(* Logix 5000 project; controller STAT 1756-L72 rev 20.12; software revision 20.04; part 18 of 34 *)
(* tags used below, declared in another part *)
   B14 : DINT[30];
   B16 : DINT[30];
   B17 : DINT[30];
   B3 : DINT[256];
   B9 : DINT[40];
   F8 : REAL[256];
   I1_005_Bit15 : ALIAS FOR I1[5].15;
   I6_001_Bit07 : ALIAS FOR I6[1].7;   // pulse debietmeter zandfilter osmose
   I7_000_Bit08 : ALIAS FOR I7[0].8;   // midden alarm ketel tampon
   N12 : DINT[230];
   N13 : DINT[230];
   N26 : DINT[256];
   O12_001_Bit14 : ALIAS FOR O12[1].14;   // STFA1_EV1 STFA1_EV1
   O12_001_Bit15 : ALIAS FOR O12[1].15;   // STFA1_EV2 STFA1_EV2
   O13_000_Bit00 : ALIAS FOR O13[0].0;   // STFA1_EV3 STFA1_EV3
   O13_000_Bit01 : ALIAS FOR O13[0].1;   // STFA1_EV4 STFA1_EV4
   O13_000_Bit02 : ALIAS FOR O13[0].2;   // STFA1_EV5 STFA1_EV5
   O13_000_Bit03 : ALIAS FOR O13[0].3;   // STFA1_EV6 STFA1_EV6
   O15_001_Bit13 : ALIAS FOR O15[1].13;   // TFB2_1_EV1 TFB2_1_EV1
   O15_001_Bit14 : ALIAS FOR O15[1].14;   // TFB2_1_EV2 TFB2_1_EV2
   O15_001_Bit15 : ALIAS FOR O15[1].15;   // TFB2_1_EV3 TFB2_1_EV3
   STEP_DUALM_3_4_5_6 : BOOL;
   STEP_NASPOEL_1_ET_2 : BOOL;
   T27 : TIMER[100];
   T4 : TIMER[200];
(* ibt, continued *)

ROUTINE _20_SEQ_VERZ1   (* ladder *)
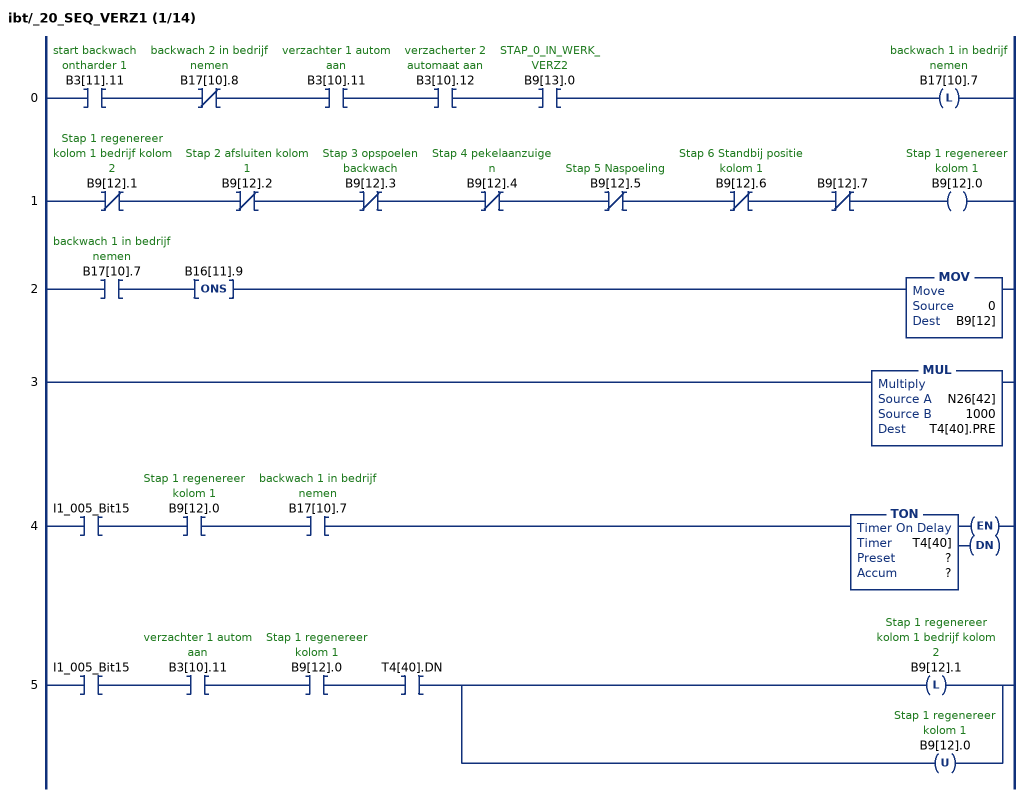
   0: XIC(B3[11].11)XIO(B17[10].8)XIC(B3[10].11)XIC(B3[10].12)XIC(B9[13].0)OTL(B17[10].7);
   1: XIO(B9[12].1)XIO(B9[12].2)XIO(B9[12].3)XIO(B9[12].4)XIO(B9[12].5)XIO(B9[12].6)XIO(B9[12].7)OTE(B9[12].0);
   2: XIC(B17[10].7)ONS(B16[11].9)MOV(0,B9[12]);
   3: MUL(N26[42],1000,T4[40].PRE);
   4: XIC(I1_005_Bit15)XIC(B9[12].0)XIC(B17[10].7)TON(T4[40],?,?);
   5: XIC(I1_005_Bit15)XIC(B3[10].11)XIC(B9[12].0)XIC(T4[40].DN)[OTL(B9[12].1) ,OTU(B9[12].0) ];
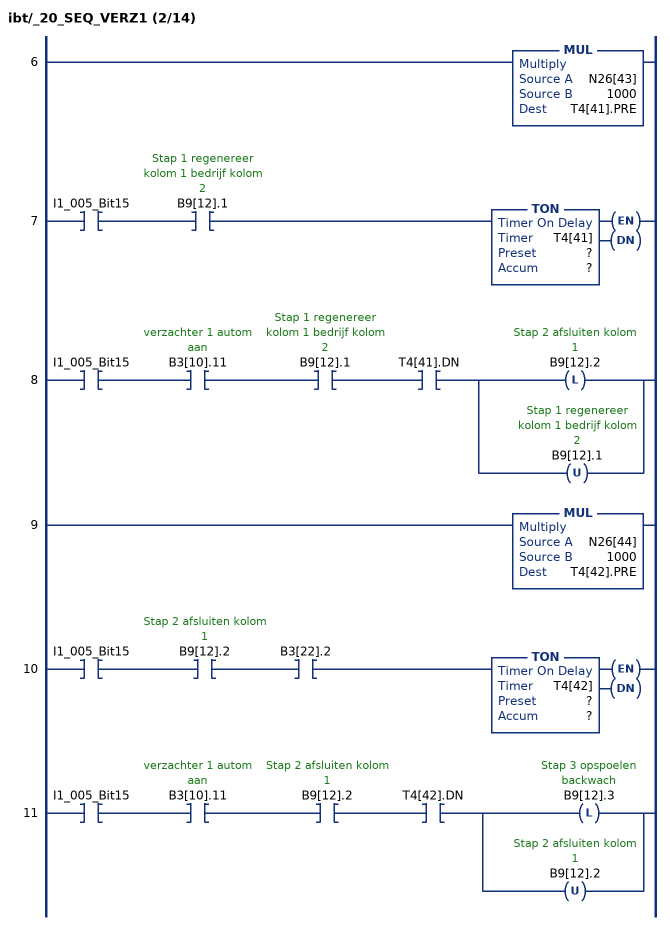
   6: MUL(N26[43],1000,T4[41].PRE);
   7: XIC(I1_005_Bit15)XIC(B9[12].1)TON(T4[41],?,?);
   8: XIC(I1_005_Bit15)XIC(B3[10].11)XIC(B9[12].1)XIC(T4[41].DN)[OTL(B9[12].2) ,OTU(B9[12].1) ];
   9: MUL(N26[44],1000,T4[42].PRE);
   10: XIC(I1_005_Bit15)XIC(B9[12].2)XIC(B3[22].2)TON(T4[42],?,?);
   11: XIC(I1_005_Bit15)XIC(B3[10].11)XIC(B9[12].2)XIC(T4[42].DN)[OTL(B9[12].3) ,OTU(B9[12].2) ];
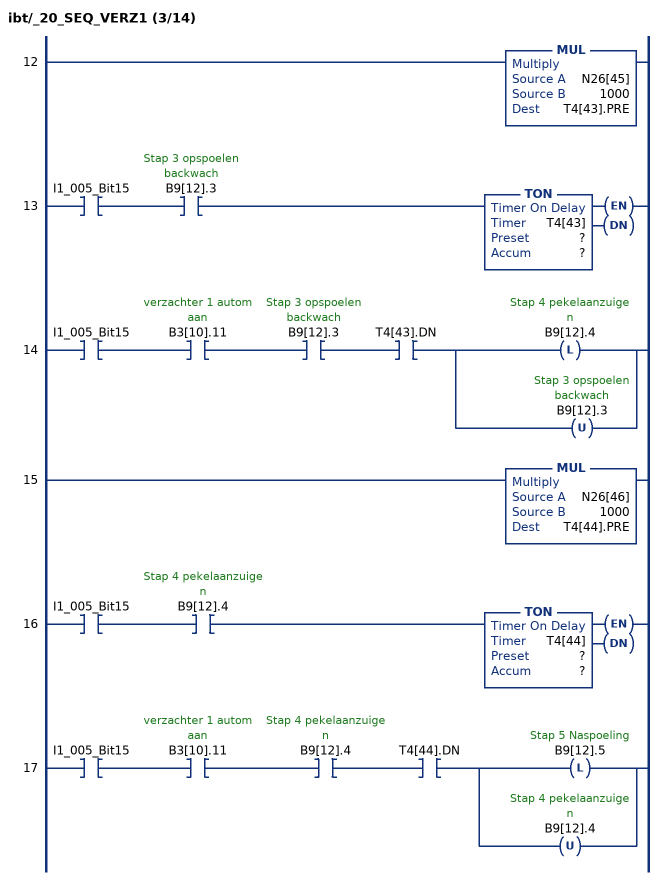
   12: MUL(N26[45],1000,T4[43].PRE);
   13: XIC(I1_005_Bit15)XIC(B9[12].3)TON(T4[43],?,?);
   14: XIC(I1_005_Bit15)XIC(B3[10].11)XIC(B9[12].3)XIC(T4[43].DN)[OTL(B9[12].4) ,OTU(B9[12].3) ];
   15: MUL(N26[46],1000,T4[44].PRE);
   16: XIC(I1_005_Bit15)XIC(B9[12].4)TON(T4[44],?,?);
   17: XIC(I1_005_Bit15)XIC(B3[10].11)XIC(B9[12].4)XIC(T4[44].DN)[OTL(B9[12].5) ,OTU(B9[12].4) ];
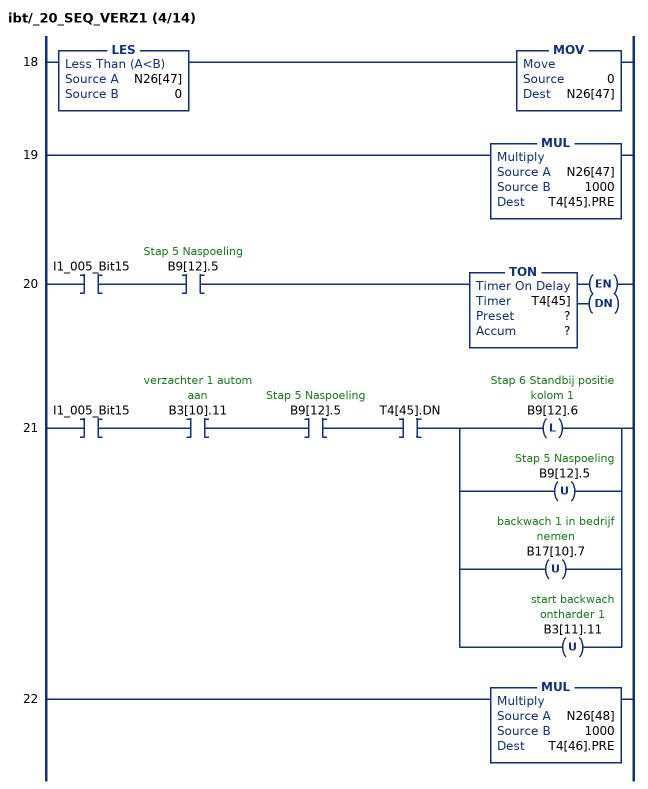
   18: LES(N26[47],0)MOV(0,N26[47]);
   19: MUL(N26[47],1000,T4[45].PRE);
   20: XIC(I1_005_Bit15)XIC(B9[12].5)TON(T4[45],?,?);
   21: XIC(I1_005_Bit15)XIC(B3[10].11)XIC(B9[12].5)XIC(T4[45].DN)[OTL(B9[12].6) ,[OTU(B9[12].5) ,[OTU(B17[10].7) ,OTU(B3[11].11) ] ] ];
   22: MUL(N26[48],1000,T4[46].PRE);
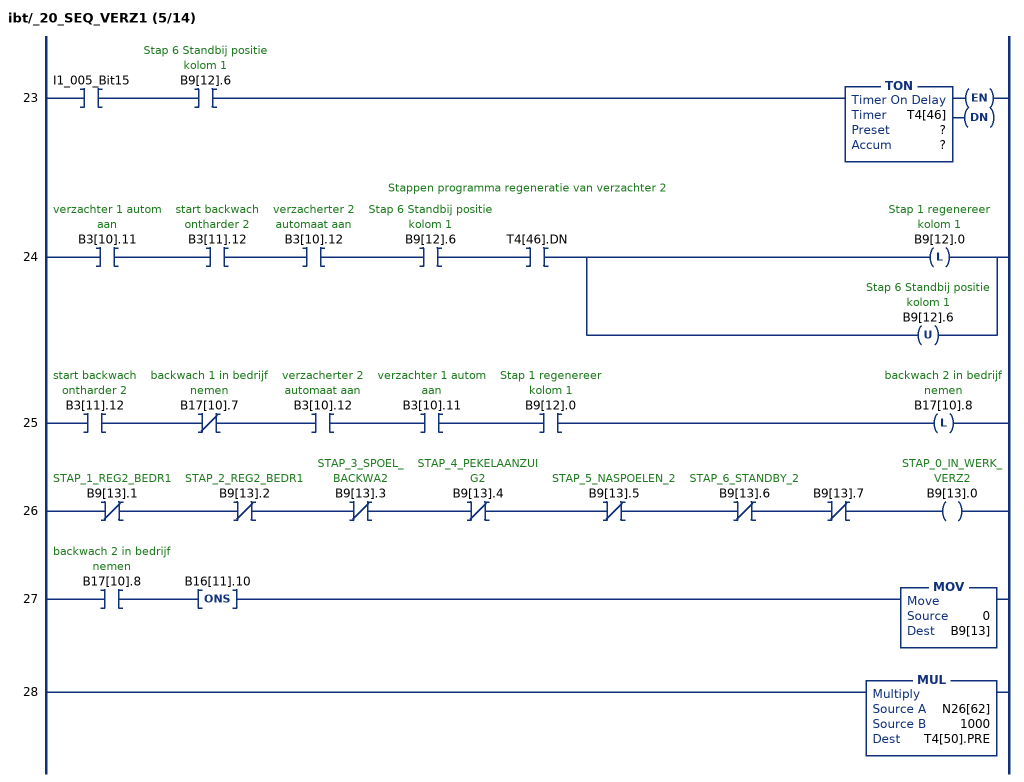
   23: XIC(I1_005_Bit15)XIC(B9[12].6)TON(T4[46],?,?);
   // Stappen programma regeneratie van verzachter 2
   24: XIC(B3[10].11)XIC(B3[11].12)XIC(B3[10].12)XIC(B9[12].6)XIC(T4[46].DN)[OTL(B9[12].0) ,OTU(B9[12].6) ];
   25: XIC(B3[11].12)XIO(B17[10].7)XIC(B3[10].12)XIC(B3[10].11)XIC(B9[12].0)OTL(B17[10].8);
   26: XIO(B9[13].1)XIO(B9[13].2)XIO(B9[13].3)XIO(B9[13].4)XIO(B9[13].5)XIO(B9[13].6)XIO(B9[13].7)OTE(B9[13].0);
   27: XIC(B17[10].8)ONS(B16[11].10)MOV(0,B9[13]);
   28: MUL(N26[62],1000,T4[50].PRE);
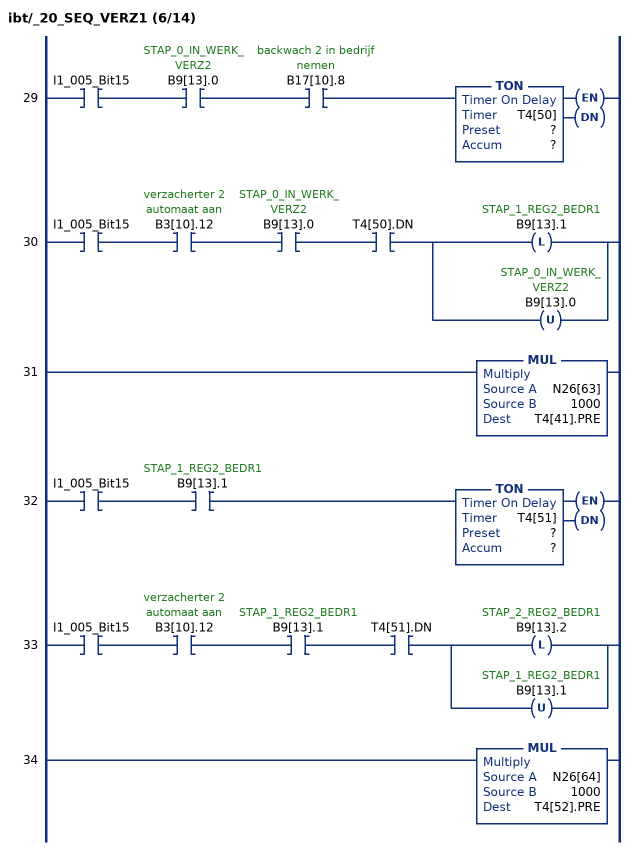
   29: XIC(I1_005_Bit15)XIC(B9[13].0)XIC(B17[10].8)TON(T4[50],?,?);
   30: XIC(I1_005_Bit15)XIC(B3[10].12)XIC(B9[13].0)XIC(T4[50].DN)[OTL(B9[13].1) ,OTU(B9[13].0) ];
   31: MUL(N26[63],1000,T4[41].PRE);
   32: XIC(I1_005_Bit15)XIC(B9[13].1)TON(T4[51],?,?);
   33: XIC(I1_005_Bit15)XIC(B3[10].12)XIC(B9[13].1)XIC(T4[51].DN)[OTL(B9[13].2) ,OTU(B9[13].1) ];
   34: MUL(N26[64],1000,T4[52].PRE);
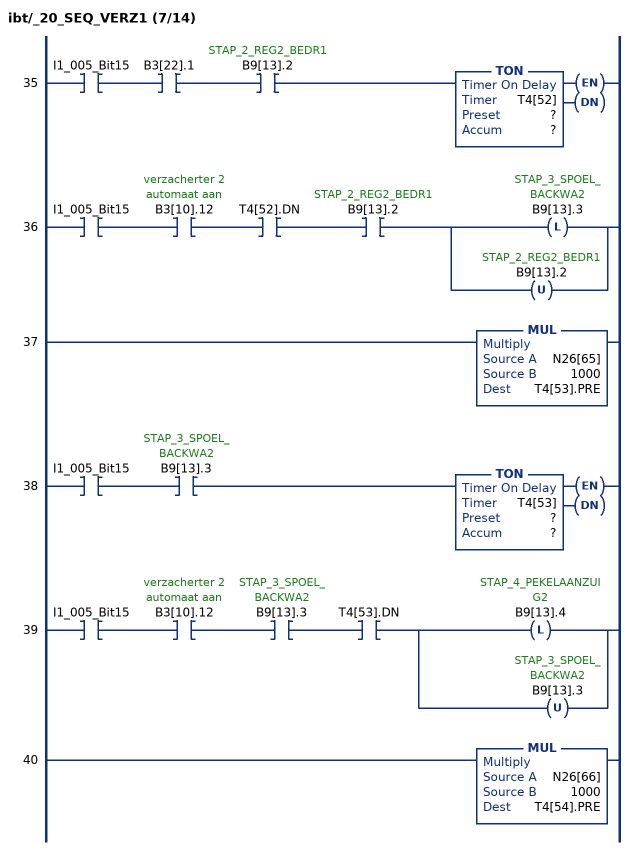
   35: XIC(I1_005_Bit15)XIC(B3[22].1)XIC(B9[13].2)TON(T4[52],?,?);
   36: XIC(I1_005_Bit15)XIC(B3[10].12)XIC(T4[52].DN)XIC(B9[13].2)[OTL(B9[13].3) ,OTU(B9[13].2) ];
   37: MUL(N26[65],1000,T4[53].PRE);
   38: XIC(I1_005_Bit15)XIC(B9[13].3)TON(T4[53],?,?);
   39: XIC(I1_005_Bit15)XIC(B3[10].12)XIC(B9[13].3)XIC(T4[53].DN)[OTL(B9[13].4) ,OTU(B9[13].3) ];
   40: MUL(N26[66],1000,T4[54].PRE);
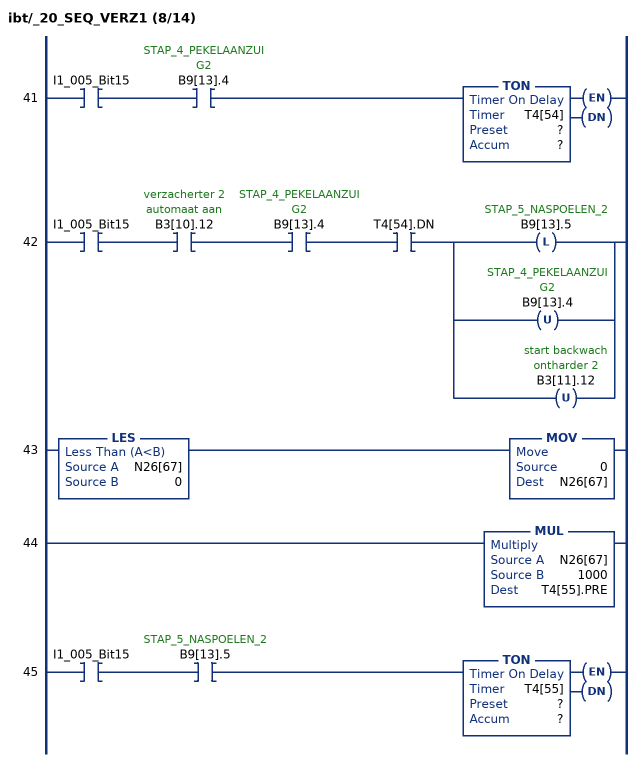
   41: XIC(I1_005_Bit15)XIC(B9[13].4)TON(T4[54],?,?);
   42: XIC(I1_005_Bit15)XIC(B3[10].12)XIC(B9[13].4)XIC(T4[54].DN)[OTL(B9[13].5) ,[OTU(B9[13].4) ,OTU(B3[11].12) ] ];
   43: LES(N26[67],0)MOV(0,N26[67]);
   44: MUL(N26[67],1000,T4[55].PRE);
   45: XIC(I1_005_Bit15)XIC(B9[13].5)TON(T4[55],?,?);
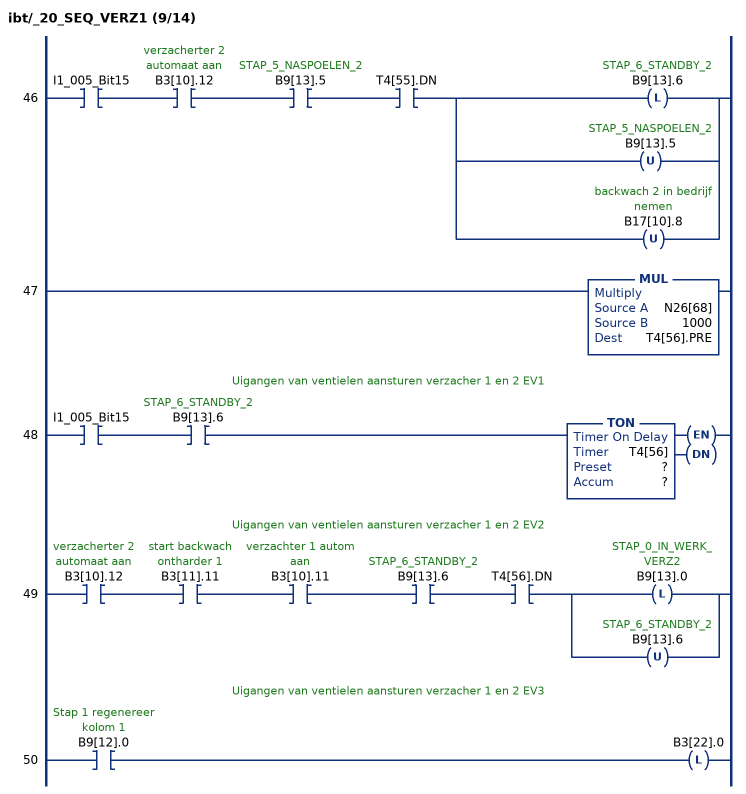
   46: XIC(I1_005_Bit15)XIC(B3[10].12)XIC(B9[13].5)XIC(T4[55].DN)[OTL(B9[13].6) ,[OTU(B9[13].5) ,OTU(B17[10].8) ] ];
   47: MUL(N26[68],1000,T4[56].PRE);
   // Uigangen van ventielen aansturen verzacher 1 en 2 EV1
   48: XIC(I1_005_Bit15)XIC(B9[13].6)TON(T4[56],?,?);
   // Uigangen van ventielen aansturen verzacher 1 en 2 EV2
   49: XIC(B3[10].12)XIC(B3[11].11)XIC(B3[10].11)XIC(B9[13].6)XIC(T4[56].DN)[OTL(B9[13].0) ,OTU(B9[13].6) ];
   // Uigangen van ventielen aansturen verzacher 1 en 2 EV3
   50: XIC(B9[12].0)OTL(B3[22].0);
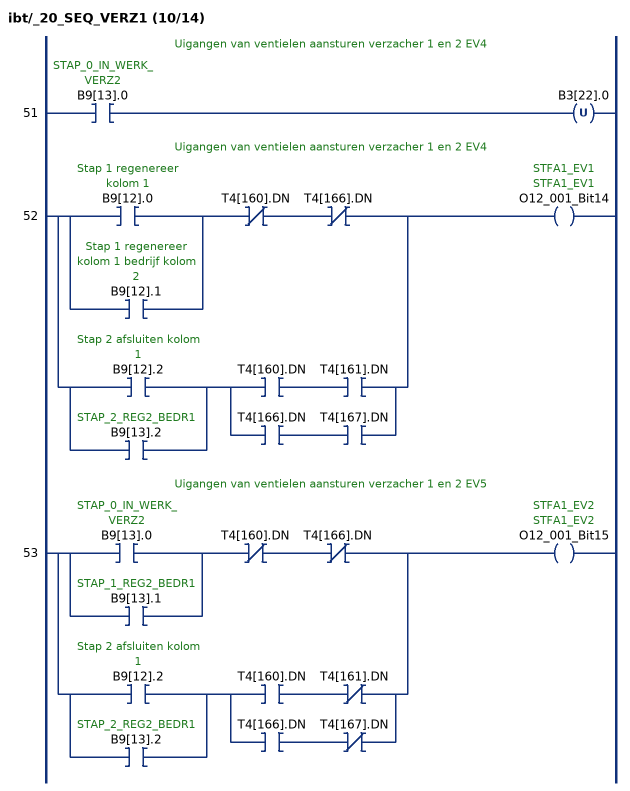
   // Uigangen van ventielen aansturen verzacher 1 en 2 EV4
   51: XIC(B9[13].0)OTU(B3[22].0);
   // Uigangen van ventielen aansturen verzacher 1 en 2 EV4
   52: [[XIC(B9[12].0) ,XIC(B9[12].1) ] XIO(T4[160].DN) XIO(T4[166].DN) ,[XIC(B9[12].2) ,XIC(B9[13].2) ] [XIC(T4[160].DN) XIC(T4[161].DN) ,XIC(T4[166].DN) XIC(T4[167].DN) ] ]OTE(O12_001_Bit14);
   // Uigangen van ventielen aansturen verzacher 1 en 2 EV5
   53: [[XIC(B9[13].0) ,XIC(B9[13].1) ] XIO(T4[160].DN) XIO(T4[166].DN) ,[XIC(B9[12].2) ,XIC(B9[13].2) ] [XIC(T4[160].DN) XIO(T4[161].DN) ,XIC(T4[166].DN) XIO(T4[167].DN) ] ]OTE(O12_001_Bit15);
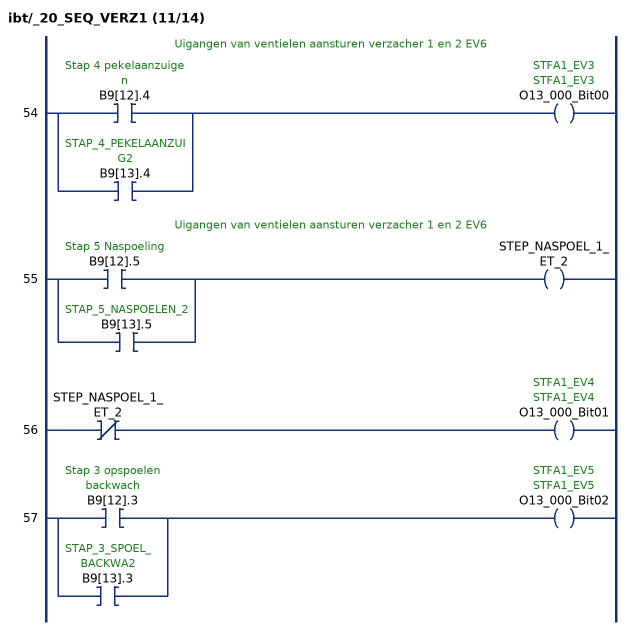
   // Uigangen van ventielen aansturen verzacher 1 en 2 EV6
   54: [XIC(B9[12].4) ,XIC(B9[13].4) ]OTE(O13_000_Bit00);
   // Uigangen van ventielen aansturen verzacher 1 en 2 EV6
   55: [XIC(B9[12].5) ,XIC(B9[13].5) ]OTE(STEP_NASPOEL_1_ET_2);
   56: XIO(STEP_NASPOEL_1_ET_2)OTE(O13_000_Bit01);
   57: [XIC(B9[12].3) ,XIC(B9[13].3) ]OTE(O13_000_Bit02);
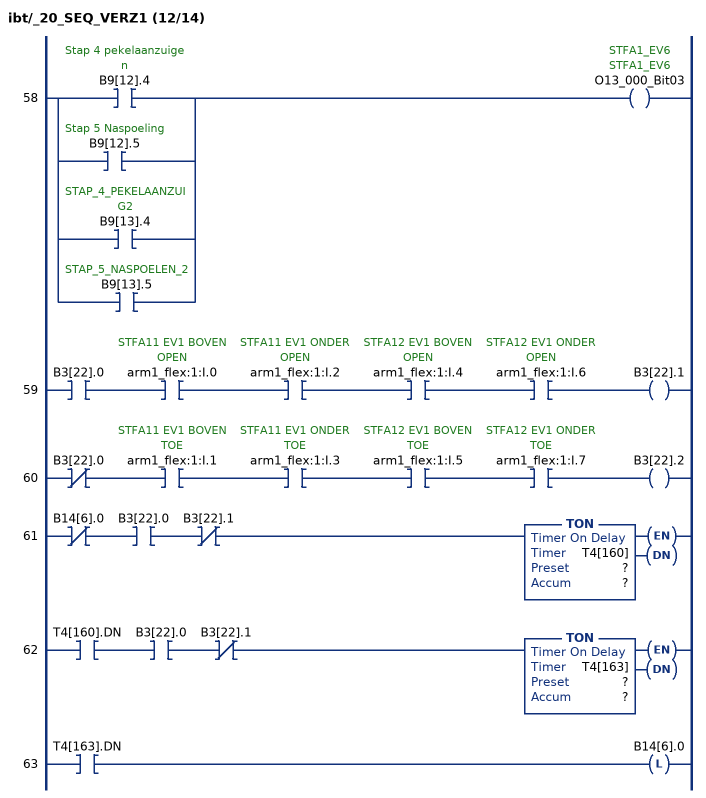
   58: [XIC(B9[12].4) ,[XIC(B9[12].5) ,[XIC(B9[13].4) ,XIC(B9[13].5) ] ] ]OTE(O13_000_Bit03);
   59: XIC(B3[22].0)XIC(arm1_flex:1:I.0)XIC(arm1_flex:1:I.2)XIC(arm1_flex:1:I.4)XIC(arm1_flex:1:I.6)OTE(B3[22].1);
   60: XIO(B3[22].0)XIC(arm1_flex:1:I.1)XIC(arm1_flex:1:I.3)XIC(arm1_flex:1:I.5)XIC(arm1_flex:1:I.7)OTE(B3[22].2);
   61: XIO(B14[6].0)XIC(B3[22].0)XIO(B3[22].1)TON(T4[160],?,?);
   62: XIC(T4[160].DN)XIC(B3[22].0)XIO(B3[22].1)TON(T4[163],?,?);
   63: XIC(T4[163].DN)OTL(B14[6].0);
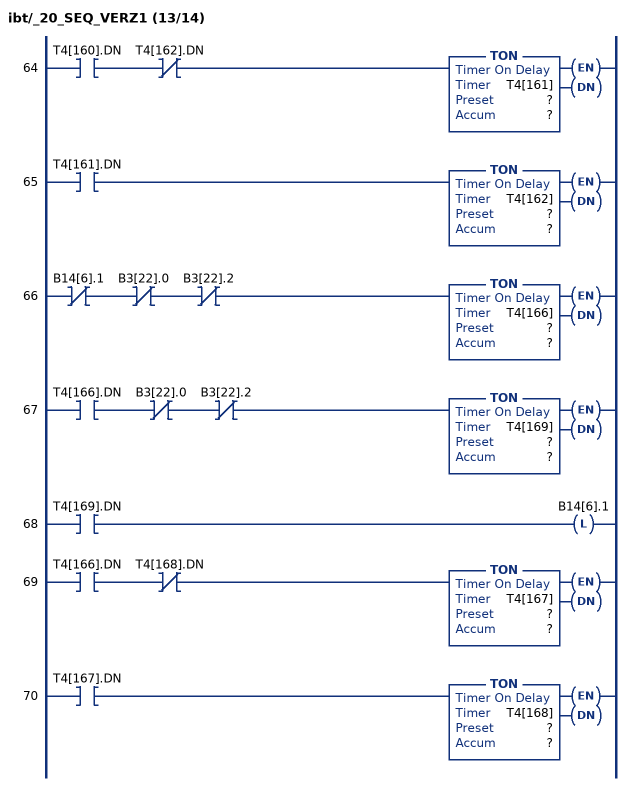
   64: XIC(T4[160].DN)XIO(T4[162].DN)TON(T4[161],?,?);
   65: XIC(T4[161].DN)TON(T4[162],?,?);
   66: XIO(B14[6].1)XIO(B3[22].0)XIO(B3[22].2)TON(T4[166],?,?);
   67: XIC(T4[166].DN)XIO(B3[22].0)XIO(B3[22].2)TON(T4[169],?,?);
   68: XIC(T4[169].DN)OTL(B14[6].1);
   69: XIC(T4[166].DN)XIO(T4[168].DN)TON(T4[167],?,?);
   70: XIC(T4[167].DN)TON(T4[168],?,?);
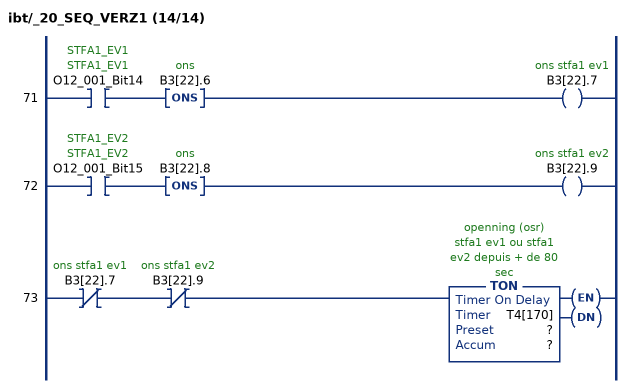
   71: XIC(O12_001_Bit14)ONS(B3[22].6)OTE(B3[22].7);
   72: XIC(O12_001_Bit15)ONS(B3[22].8)OTE(B3[22].9);
   73: XIO(B3[22].7)XIO(B3[22].9)TON(T4[170],?,?);
END_ROUTINE

ROUTINE _21_SEQ_DBLMED   (* ladder *)
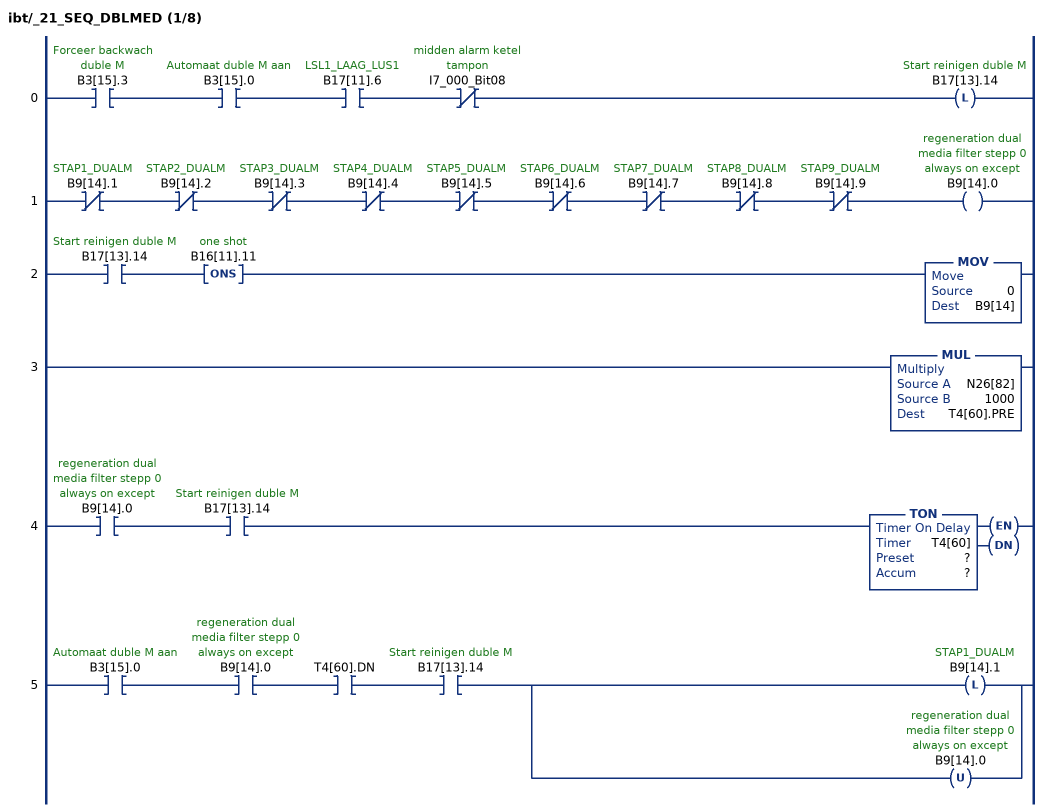
   0: XIC(B3[15].3)XIC(B3[15].0)XIC(B17[11].6)XIO(I7_000_Bit08)OTL(B17[13].14);
   1: XIO(B9[14].1)XIO(B9[14].2)XIO(B9[14].3)XIO(B9[14].4)XIO(B9[14].5)XIO(B9[14].6)XIO(B9[14].7)XIO(B9[14].8)XIO(B9[14].9)OTE(B9[14].0);
   2: XIC(B17[13].14)ONS(B16[11].11)MOV(0,B9[14]);
   3: MUL(N26[82],1000,T4[60].PRE);
   4: XIC(B9[14].0)XIC(B17[13].14)TON(T4[60],?,?);
   5: XIC(B3[15].0)XIC(B9[14].0)XIC(T4[60].DN)XIC(B17[13].14)[OTL(B9[14].1) ,OTU(B9[14].0) ];
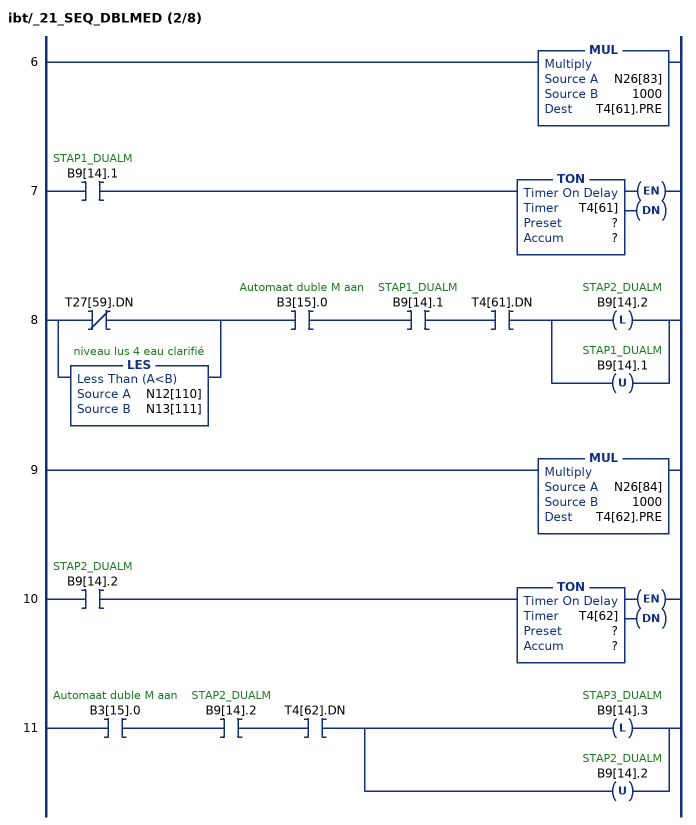
   6: MUL(N26[83],1000,T4[61].PRE);
   7: XIC(B9[14].1)TON(T4[61],?,?);
   8: [XIO(T27[59].DN) ,LES(N12[110],N13[111]) ]XIC(B3[15].0)XIC(B9[14].1)XIC(T4[61].DN)[OTL(B9[14].2) ,OTU(B9[14].1) ];
   9: MUL(N26[84],1000,T4[62].PRE);
   10: XIC(B9[14].2)TON(T4[62],?,?);
   11: XIC(B3[15].0)XIC(B9[14].2)XIC(T4[62].DN)[OTL(B9[14].3) ,OTU(B9[14].2) ];
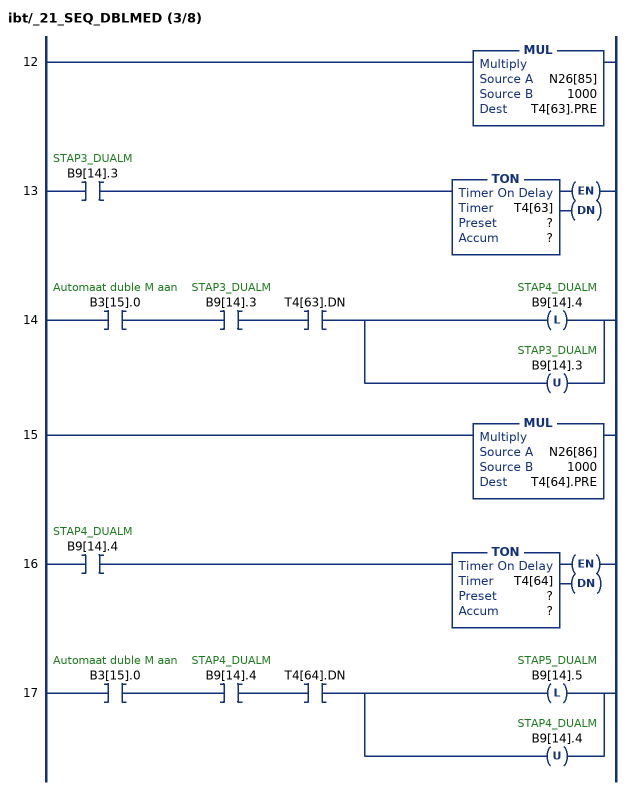
   12: MUL(N26[85],1000,T4[63].PRE);
   13: XIC(B9[14].3)TON(T4[63],?,?);
   14: XIC(B3[15].0)XIC(B9[14].3)XIC(T4[63].DN)[OTL(B9[14].4) ,OTU(B9[14].3) ];
   15: MUL(N26[86],1000,T4[64].PRE);
   16: XIC(B9[14].4)TON(T4[64],?,?);
   17: XIC(B3[15].0)XIC(B9[14].4)XIC(T4[64].DN)[OTL(B9[14].5) ,OTU(B9[14].4) ];
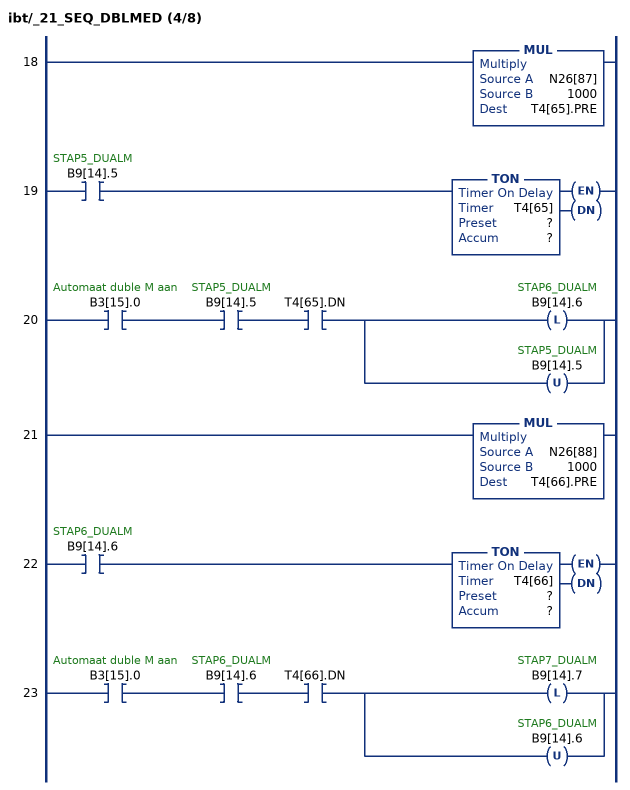
   18: MUL(N26[87],1000,T4[65].PRE);
   19: XIC(B9[14].5)TON(T4[65],?,?);
   20: XIC(B3[15].0)XIC(B9[14].5)XIC(T4[65].DN)[OTL(B9[14].6) ,OTU(B9[14].5) ];
   21: MUL(N26[88],1000,T4[66].PRE);
   22: XIC(B9[14].6)TON(T4[66],?,?);
   23: XIC(B3[15].0)XIC(B9[14].6)XIC(T4[66].DN)[OTL(B9[14].7) ,OTU(B9[14].6) ];
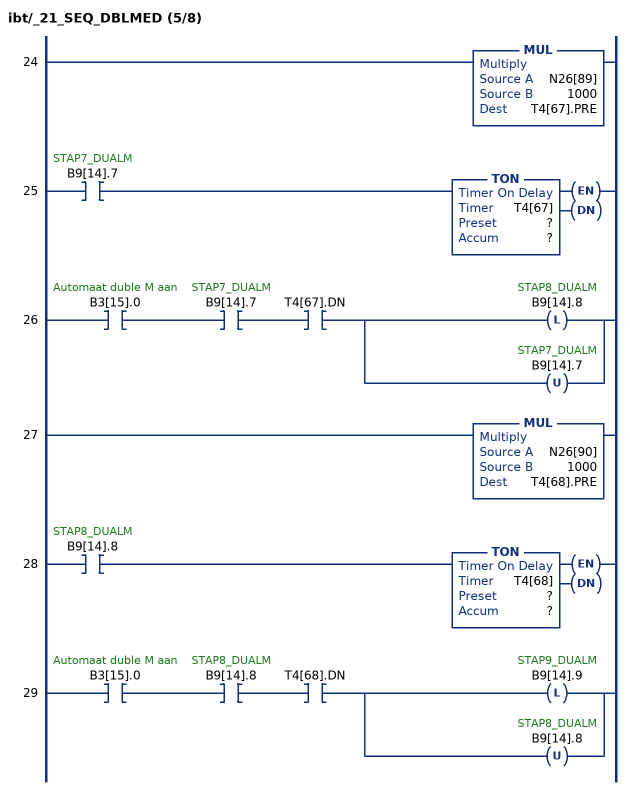
   24: MUL(N26[89],1000,T4[67].PRE);
   25: XIC(B9[14].7)TON(T4[67],?,?);
   26: XIC(B3[15].0)XIC(B9[14].7)XIC(T4[67].DN)[OTL(B9[14].8) ,OTU(B9[14].7) ];
   27: MUL(N26[90],1000,T4[68].PRE);
   28: XIC(B9[14].8)TON(T4[68],?,?);
   29: XIC(B3[15].0)XIC(B9[14].8)XIC(T4[68].DN)[OTL(B9[14].9) ,OTU(B9[14].8) ];
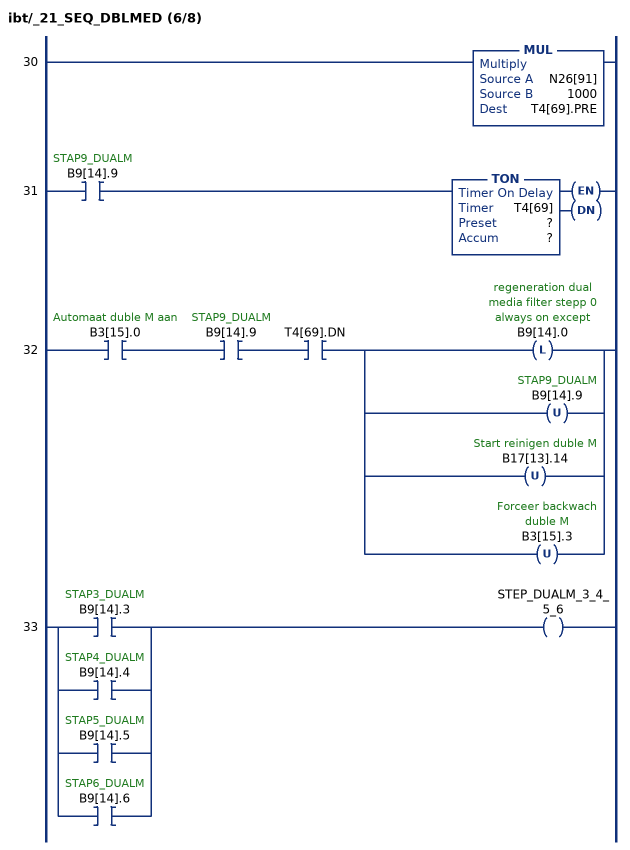
   30: MUL(N26[91],1000,T4[69].PRE);
   31: XIC(B9[14].9)TON(T4[69],?,?);
   32: XIC(B3[15].0)XIC(B9[14].9)XIC(T4[69].DN)[OTL(B9[14].0) ,[OTU(B9[14].9) ,[OTU(B17[13].14) ,OTU(B3[15].3) ] ] ];
   33: [XIC(B9[14].3) ,[XIC(B9[14].4) ,[XIC(B9[14].5) ,XIC(B9[14].6) ] ] ]OTE(STEP_DUALM_3_4_5_6);
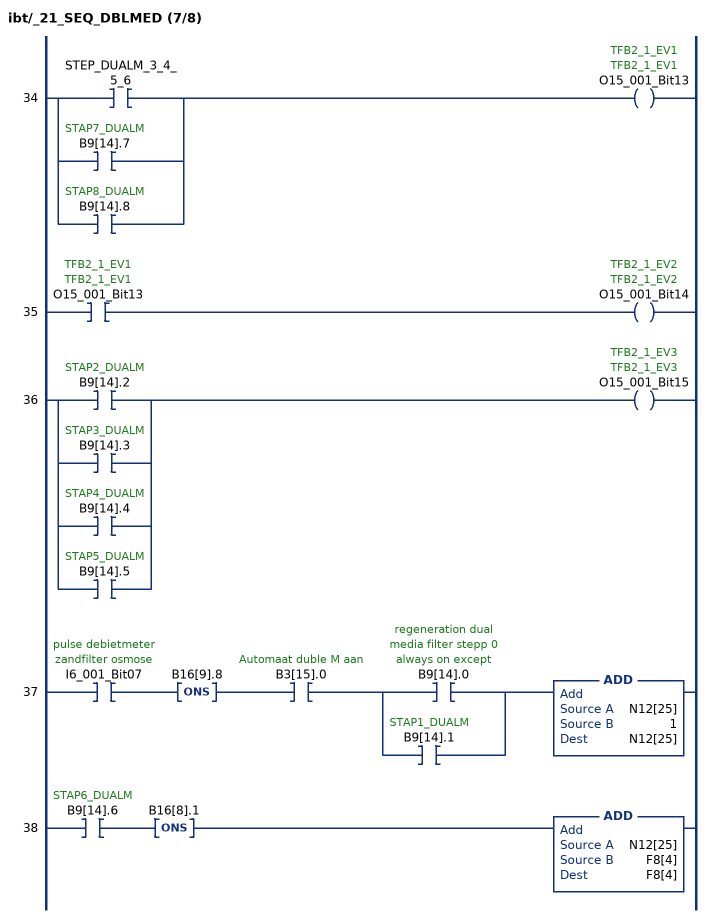
   34: [XIC(STEP_DUALM_3_4_5_6) ,[XIC(B9[14].7) ,XIC(B9[14].8) ] ]OTE(O15_001_Bit13);
   35: XIC(O15_001_Bit13)OTE(O15_001_Bit14);
   36: [XIC(B9[14].2) ,[XIC(B9[14].3) ,[XIC(B9[14].4) ,XIC(B9[14].5) ] ] ]OTE(O15_001_Bit15);
   37: XIC(I6_001_Bit07)ONS(B16[9].8)XIC(B3[15].0)[XIC(B9[14].0) ,XIC(B9[14].1) ]ADD(N12[25],1,N12[25]);
   38: XIC(B9[14].6)ONS(B16[8].1)ADD(N12[25],F8[4],F8[4]);
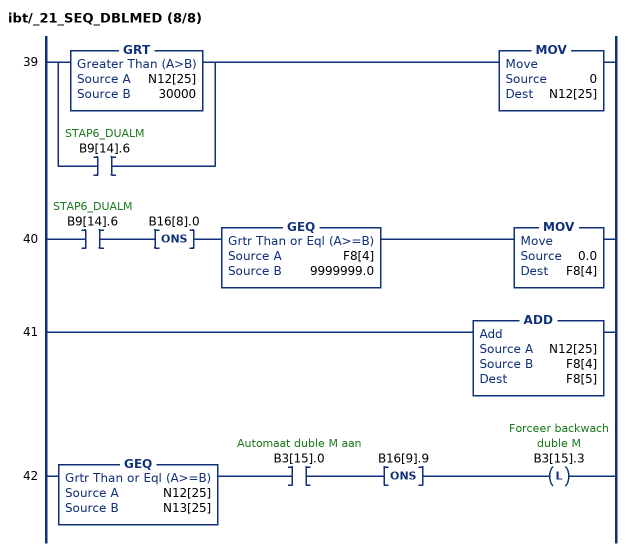
   39: [GRT(N12[25],30000) ,XIC(B9[14].6) ]MOV(0,N12[25]);
   40: XIC(B9[14].6)ONS(B16[8].0)GEQ(F8[4],9999999.0)MOV(0.0,F8[4]);
   41: ADD(N12[25],F8[4],F8[5]);
   42: GEQ(N12[25],N13[25])XIC(B3[15].0)ONS(B16[9].9)OTL(B3[15].3);
END_ROUTINE
